(* CODESYS project FillingCappingSol_Version9.project

Project tree, tasks and I/O mapping:
  Device : CODESYS Control Win V3, 3S - Smart Software Solutions GmbH, order no. 305021, version 3.5.9.40
    application Application
      libraries: Standard, * (System)
      task MainTask (cyclic, interval t#10ms, priority 1) calls GEMMA, OutputWrite
      program F1_NormalProduction [ST]
      program D3_ProductionWithFailures [ST]
      program F2_StartingProcedure [ST]
      program F3_FinishingProcedure [ST]
      program F4_StationProducingTest [ST]
      program F5_OrderedProducingTest [ST]
      program GEMMA [ST]
      program OutputWrite [ST]
      global variables GVL
      Symbols
*)

// Device/Application/GVL
{attribute 'qualified_only'}
VAR_GLOBAL

//INPUTS
	
	//Sensors
	a0:BOOL:=FALSE;	
	a1:BOOL:=FALSE;
	b0:BOOL:=FALSE;	
	b1:BOOL:=FALSE;
	c0:BOOL:=FALSE;	
	c1:BOOL:=FALSE;
	e0:BOOL:=FALSE;	
	e1:BOOL:=FALSE;
	e2:BOOL:=FALSE;
	g0:BOOL:=FALSE;	
	g1:BOOL:=FALSE;	
	h0:BOOL:=FALSE;	
	h1:BOOL:=FALSE;	
	CP1:BOOL:=FALSE;
	CP2:BOOL:=FALSE;
	CP3:BOOL:=FALSE;	
	
	//Commands
	Mode:UINT:=0; //selector
	A:BOOL:=FALSE; //automatic
	SA:BOOL:=FALSE; //semi-automatic
	MA:BOOL:=FALSE; //manual	
	START:BOOL:=FALSE; //start PB
	PE:BOOL:=TRUE; //emergency interrupter
	STOP:BOOL:=TRUE; //stop PB	
	EM:BOOL:=FALSE; //Empty Machine
	TM:BOOL:=FALSE; //Manual Capping
	ST_:BOOL:=FALSE; //Operating Test
	CR:BOOL:=FALSE; //Capping Repaired
	OC:BOOL:=FALSE; //Operator Check
	MMC:BOOL:=FALSE; //Manual Movement Check
	
	//Semi-automatic
	Station:UINT:=0; //selector
	Station1:BOOL:=FALSE;
	Station2:BOOL:=FALSE;
	Station3:BOOL:=FALSE;
	SC:BOOL:=FALSE; //start cycle
	
	//Manual
	a_p_manual:BOOL:=FALSE; //a+
	a_m_manual:BOOL:=FALSE; //a-
	b_p_manual:BOOL:=FALSE; //b+
	b_m_manual:BOOL:=FALSE; //b-
	c_p_manual:BOOL:=FALSE; //c+
	c_m_manual:BOOL:=FALSE; //c-
	e_p_manual:BOOL:=FALSE; //e+
	g_p_manual:BOOL:=FALSE; //g+
	g_m_manual:BOOL:=FALSE; //g-
	d_p_manual:BOOL:=FALSE; //d+
	f_p_manual:BOOL:=FALSE; //f+	
	h_p_manual:BOOL:=FALSE; //h+
	h_m_manual:BOOL:=FALSE; //h-
	
	//OUTPUTS
	
	//Actuators
	a_p:BOOL:=FALSE; //a+
	a_m:BOOL:=FALSE; //a-
	b_p:BOOL:=FALSE; //b+
	b_m:BOOL:=FALSE; //b-
	c_p:BOOL:=FALSE; //c+
	c_m:BOOL:=FALSE; //c-
	e_p:BOOL:=FALSE; //e+
	g_p:BOOL:=FALSE; //g+
	g_m:BOOL:=FALSE; //g-
	d_p:BOOL:=FALSE; //d+
	f_p:BOOL:=FALSE; //f+	
	h_p:BOOL:=FALSE; //h+
	h_m:BOOL:=FALSE; //h-	
	
	//Extra
	Flag_Timer : BOOL := FALSE;
	extra2 : BOOL := FALSE;	
	Timer1 : TON;
	E_1 : BOOL := TRUE;
	E_2 : BOOL := FALSE;
	E3 : BOOL := FALSE;
	E4 : BOOL := FALSE;
	E5 : BOOL := FALSE;
	E6 : BOOL := FALSE;
	E7 : BOOL := FALSE;
	E8 : BOOL := FALSE;
	E9 : BOOL := FALSE;
	E10 : BOOL := FALSE;
	E11 : BOOL := FALSE;
	E12 : BOOL := FALSE;
	E13 : BOOL := FALSE;
	
	E20 : BOOL := TRUE;
	E21 : BOOL := FALSE;
	E22 : BOOL := FALSE;
	E23 : BOOL := FALSE;
	E24 : BOOL := FALSE;
	E25 : BOOL := FALSE;
	E26 : BOOL := FALSE;
	E27 : BOOL := FALSE;
	E28 : BOOL := FALSE;
	E29 : BOOL := FALSE;
	
	Flag_F2 : BOOL := FALSE;
	Step_Button : BOOL := FALSE;
	extra : bool := false;
END_VAR

// Device/Application/GEMMA
PROGRAM GEMMA
VAR
	State:UINT:=15;
	Flag_Entry:BOOL:=TRUE;
	RP:BOOL:=FALSE;
	
	//GEMMA states
	F1:BOOL:=FALSE;
	F2:BOOL:=FALSE;
	F3:BOOL:=FALSE;
	F4:BOOL:=FALSE;
	F5:BOOL:=FALSE;
	F6:BOOL:=FALSE;
	A1:BOOL:=FALSE;
	A2:BOOL:=FALSE;
	A3:BOOL:=FALSE;
	A4:BOOL:=FALSE;
	A5:BOOL:=FALSE;
	A6:BOOL:=FALSE;
	A7:BOOL:=FALSE;
	D1:BOOL:=FALSE;
	D2:BOOL:=FALSE;
	D3:BOOL:=FALSE;
	
	//Transitions
	T_A1_F4:BOOL:=FALSE;
	T_A1_F5:BOOL:=FALSE;
	T_A1_F2:BOOL:=FALSE;
	T_F1_D1:BOOL:=FALSE;
END_VAR

CASE State OF
	
	1:  // F1 NORMAL PRODUCTION
		IF Flag_Entry THEN
			F1:=TRUE;
			Flag_Entry:=FALSE;
		END_IF

		//Do Behavior
		F1_NormalProduction();

		T_F1_D1:=NOT GVL.PE OR F1_NormalProduction.Alarm;		
		//Exit Common Behavior
		IF T_F1_D1 OR F1_NormalProduction.T_F4 OR F1_NormalProduction.T_F5 
		OR F1_NormalProduction.T_F3 OR F1_NormalProduction.T_D3 
		OR F1_NormalProduction.T_A2 THEN
			F1:=FALSE;
			Flag_Entry:=TRUE;
		END_IF	
		//Exit Behavior
		IF T_F1_D1 THEN
			State:=7; // Transition to D1 emergency stop
			T_F1_D1:=FALSE;
		ELSIF F1_NormalProduction.T_F4 THEN
			State:=4; // Transition to F4 disordered producing test
			F1_NormalProduction.T_F4:=FALSE;
			F4_StationProducingTest.Reset:=TRUE;
 		ELSIF F1_NormalProduction.T_F5 THEN
			State:=5; // Transition to F5 ordered producing test
			F1_NormalProduction.T_F5:=FALSE;
			F5_OrderedProducingTest.Reset:=TRUE;
 		ELSIF F1_NormalProduction.T_F3 THEN
			State:=3; // Transition to F3 finishing procedure
			F1_NormalProduction.T_F3:=FALSE;
			F3_FinishingProcedure.Reset:=TRUE;
 		ELSIF F1_NormalProduction.T_D3 THEN
			State:=9; // Transition to D3 production with failure
			F1_NormalProduction.T_D3:=FALSE;
 		ELSIF F1_NormalProduction.T_A2 THEN
			State:=11; // Transition to A2 end of cycle request
			F1_NormalProduction.T_A2:=FALSE;
		END_IF
	
	2:  // F2 STARTING PROCEDURE
		
		//Entry Behavior
		IF Flag_Entry THEN
			F2:=TRUE;
			Flag_Entry:=FALSE;
		END_IF
		
		//During Behavior
		F2_StartingProcedure();
	
		//Exit Common Behavior
		IF F2_StartingProcedure.F2_DN OR NOT GVL.PE THEN
			F2:=FALSE;
			Flag_Entry:=TRUE;
		END_IF
		//Exit Behavior	
		IF NOT GVL.PE THEN
			State:=7; // Transition to D1 emergency stop
		ELSIF F2_StartingProcedure.F2_DN THEN
			State:=1; // Transition to F1 normal production
			F2_StartingProcedure.F2_DN:=FALSE;
			F1_NormalProduction.Reset:=TRUE;
		END_IF

	3:  // F3 FINISHING PROCEDURE

		//Entry Behavior
		IF Flag_Entry THEN
			F3:=TRUE;
			Flag_Entry:=FALSE;
		END_IF
		
		//Do Behavior
		F3_FinishingProcedure();

		//Exit Behavior
		IF F3_FinishingProcedure.F3_DN OR NOT GVL.PE THEN
			F3:=FALSE;
			Flag_Entry:=TRUE;
		END_IF	
		IF NOT GVL.PE THEN
			State:=7; // Transition to D1 emergency stop
		ELSIF F3_FinishingProcedure.F3_DN THEN
			State:=10; // Transition to A1 stopped at initial state
			F3_FinishingProcedure.F3_DN:=FALSE;
		END_IF
	
	4:  // F4 DISORDERED PRODUCING TEST

		//Entry Behavior
		IF Flag_Entry THEN
			F4:=TRUE;
			Flag_Entry:=FALSE;
		END_IF
		
		//Do Behavior
		F4_StationProducingTest();

		//Exit Behavior
		IF GVL.MA OR NOT GVL.PE THEN
			F4:=FALSE;
			Flag_Entry:=TRUE;
		END_IF	
		IF NOT GVL.PE THEN
			State:=7; // Transition to D1 emergency stop
		ELSIF GVL.MA THEN
			State:=15; // Transition to A6 restarting
		END_IF	

	5:  // F5 ORDERED PRODUCING TEST

		//Entry Behavior
		IF Flag_Entry THEN
			F5:=TRUE;
			Flag_Entry:=FALSE;
		END_IF
		
		//Do Behavior
		F5_OrderedProducingTest();

		//Exit Behavior
		IF F5_OrderedProducingTest.T_F1 OR F5_OrderedProducingTest.T_F4 OR NOT GVL.PE THEN
			F5:=FALSE;
			Flag_Entry:=TRUE;
		END_IF	
		IF NOT GVL.PE THEN
			State:=7; // Transition to D1 emergency stop		
		ELSIF F5_OrderedProducingTest.T_F1 THEN
			State:=1; // Transition to F1 normal production
			F5_OrderedProducingTest.T_F1:=FALSE;
			F1_NormalProduction.PreviousStateF5:=TRUE;
			F1_NormalProduction.Reset:=TRUE;
		ELSIF F5_OrderedProducingTest.T_F4 THEN
			State:=4; // Transition to F4 disordered producing test
			F5_OrderedProducingTest.T_F4:=FALSE;
			F4_StationProducingTest.Reset:=TRUE;
		END_IF
	
	6:  // F6 OPERATING TEST
	
	7:  // D1 EMERGENCY STOP

		//Entry Behavior
		IF Flag_Entry THEN
			D1:=TRUE;
			Flag_Entry:=FALSE;
		END_IF

		//Do Behavior
		RP:=GVL.h0 AND GVL.b0 AND GVL.a0 AND GVL.c0 AND NOT GVL.d_p AND NOT GVL.e_p AND NOT GVL.f_p AND GVL.g0;
		
		//Exit Behavior
		IF GVL.PE AND RP THEN
			D1:=FALSE;
			Flag_Entry:=TRUE;
			State:=14;   // Transition to A5 preparation for restarging after a failure
		END_IF	 
	
	8:  // D2 DIAGNOSIS AND TREATMENT OF FAILURES

		//Entry Behavior
		IF Flag_Entry THEN
			D2:=TRUE;
			Flag_Entry:=FALSE;
		END_IF

		//Do Behavior
		
		//Exit Behavior
		IF GVL.CR THEN
			D2:=FALSE;
			Flag_Entry:=TRUE;
			State:=14;   // Transition to A5 preparation for restarging after a failure
		END_IF	 
	
	9:  // D3 PRODUCTION WITH FAILURES

		//Entry Behavior
		IF Flag_Entry THEN
			D3:=TRUE;
			Flag_Entry:=FALSE;
		END_IF

		//Do Behavior
		D3_ProductionWithFailures();
		
		//Exit Behavior
		IF NOT GVL.TM THEN
			D3:=FALSE;
			Flag_Entry:=TRUE;
			State:=8;        // Transition to D2 diagnosis and treatment of failures
		END_IF	 
	
	10: // A1 STOPPED AT INITIAL STATE

		//Entry Behavior
		IF Flag_Entry THEN
			A1:=TRUE;
			Flag_Entry:=FALSE;
		END_IF

		//Do Behavior
		
		T_A1_F2:=GVL.START AND GVL.A;
		T_A1_F4:=GVL.START AND (GVL.MA OR GVL.ST_);
		T_A1_F5:=GVL.START AND GVL.SA;
		//Exit Behavior
		IF T_A1_F2 OR T_A1_F4 OR T_A1_F5 THEN
			A1:=FALSE;
			Flag_Entry:=TRUE;
		END_IF	 
		IF T_A1_F4 THEN 
			State:=4;     // Transition to F4 disordered producing test
			T_A1_F4:=FALSE;
			F4_StationProducingTest.Reset := TRUE;
		ELSIF T_A1_F5 THEN 
			State:=5;
			T_A1_F5:=FALSE;  // Transition to F5 ordered producing test
			F5_OrderedProducingTest.Reset:=TRUE;
		ELSIF T_A1_F2 THEN 
			State:=2;      // Transition to F2 starting procedure
			T_A1_F2:=FALSE; 
			F2_StartingProcedure.Reset:=TRUE;
		END_IF
			
	11: // A2 END OF CYCLE REQUEST

		//Entry Behavior
		IF Flag_Entry THEN
			A2:=TRUE;
			Flag_Entry:=FALSE;
		END_IF

		//Do Behavior
		RP:=GVL.h0 AND GVL.b0 AND GVL.a0 AND GVL.c0 AND NOT GVL.d_p AND NOT GVL.e_p AND NOT GVL.f_p AND GVL.g0;
		
		//Exit Behavior
		IF RP AND GVL.STOP	THEN
			A2:=FALSE;
			Flag_Entry:=TRUE;
			State:=10; // Transition to A1 stopped at initial state
			RP:=FALSE;
		END_IF	 
	
	12: // A3 STOP REQUESTED
	
	13: // A4 STOPPED AT A NOT-INITIAL STATE
	
	14: // A5 PREPARATION FOR RESTARTING AFTER A FAILURE

		//Entry Behavior
		IF Flag_Entry THEN
			A5:=TRUE;
			Flag_Entry:=FALSE;
		END_IF

		//Do Behavior
		
		//Exit Behavior
		IF GVL.OC THEN
			F1_NormalProduction.Alarm:=FALSE;
			A5:=FALSE;
			Flag_Entry:=TRUE;
			State:=15; // Transition to A6 restarting
		END_IF	 
	
	15: // A6 RESTARTING

		//Entry Behavior
		IF Flag_Entry THEN
			A6:=TRUE;
			Flag_Entry:=FALSE;
		END_IF

		//Do Behavior
		RP:=GVL.h0 AND GVL.b0 AND GVL.a0 AND GVL.c0 AND NOT GVL.d_p AND NOT GVL.e_p AND NOT GVL.f_p AND GVL.g0;
		
		//Exit Behavior
		IF RP AND GVL.MMC THEN
			A6:=FALSE;
			Flag_Entry:=TRUE;
			State:=10; // Transition to A1 stopped at initial state
			RP:=FALSE;
		END_IF	 
	
	16: // A7 STOPPING IN A NOT-INITIAL STATE

END_CASE

END_PROGRAM

// Device/Application/F1_NormalProduction
PROGRAM F1_NormalProduction
VAR
	State: INT;
	State2: INT;
	State3: INT;
	EM_MEM:BOOL:=FALSE;
	STOP_MEM:BOOL:=TRUE;
	CycleOver:BOOL:=FALSE;
END_VAR

VAR_INPUT
	Reset:BOOL:=FALSE;
	Alarm:BOOL:=FALSE;
	T_F4:BOOL:=FALSE;
	T_A2:BOOL:=FALSE;
	T_D3:BOOL:=FALSE;
	T_F5:BOOL:=FALSE;
	T_F3:BOOL:=FALSE;
	PreviousStateF5:BOOL:=FALSE;
END_VAR

IF (Reset) THEN
	Reset := FALSE;
	State:=3;
	State2:=0;
	State3:=0;
END_IF

IF PreviousStateF5 THEN
	PreviousStateF5:=FALSE;
	State:=1;
END_IF

CASE State OF
1:
	IF (GVL.b1 AND GVL.h1) THEN
		State := 2;
		CycleOver := FALSE;
	END_IF
2:
	IF (GVL.b0 AND GVL.h0) THEN
		State := 3;
	END_IF
3:
	IF (NOT GVL.CP1 OR NOT GVL.CP2 OR NOT GVL.CP3) THEN
		Alarm := TRUE;
	END_IF
	IF (NOT Alarm) THEN
		State := 4;
		State2 := 6;
		State3 := 8;
	END_IF
4:
	IF (GVL.a1) THEN
		State := 5;
	END_IF

END_CASE

CASE State2 OF
6:
	IF (GVL.c1) THEN
		State2 := 7;
	END_IF
END_CASE

CASE State3 OF
8:
	IF (GVL.g1) THEN
		State3 := 9;
	END_IF
9:
	IF (gvl.e1) THEN
		State3 := 10;
	END_IF
10:
	IF (GVL.g0) THEN
		State3 := 11;
	END_IF
11:
	IF (GVL.e2) THEN
		State3 := 12;
	END_IF
12:
		IF (GVL.a0 AND GVL.c0 AND GVL.e0) THEN
		State :=  1;
		State2 := 0;
		State3 := 0;
		CycleOver := TRUE;
	END_IF
END_CASE

//HMI Memory
IF GVL.EM OR NOT GVL.STOP THEN
	IF GVL.EM THEN
		EM_MEM:=TRUE;
	ELSIF NOT GVL.STOP THEN
		STOP_MEM:=FALSE;
	END_IF
END_IF 

//Exit Transition
IF CycleOver THEN
	IF NOT STOP_MEM THEN
		T_A2:=TRUE;
		STOP_MEM:=FALSE;
	ELSIF EM_MEM THEN
		T_F3:=TRUE;
		EM_MEM:=FALSE;	
	ELSIF GVL.MA OR GVL.ST_ THEN
		T_F4:=TRUE;
	ELSIF GVL.SA THEN
		T_F5:=TRUE;
	ELSIF GVL.TM THEN
		T_D3:=TRUE;
	END_IF
END_IF

END_PROGRAM

// Device/Application/F4_StationProducingTest
PROGRAM F4_StationProducingTest
VAR
	State: INT;
	State2: INT;
	State3: INT;
END_VAR

VAR_INPUT
		Reset: BOOL;
END_VAR

IF (Reset) THEN
	Reset := FALSE;
	State  := 1;
	State2 := 0;
	State3 := 0;
	IF NOT GVL.Station1 AND NOT GVL.Station3 THEN
		GVL.Station2:=TRUE;
	END_IF
END_IF


CASE State OF
1:
	IF (GVL.b1 AND GVL.h1) THEN
		State := 2;
	END_IF
2:
	IF (GVL.b0 AND GVL.h0) THEN
		State := 3;
	END_IF
3:
	IF (GVL.Station1 AND GVL.SC) THEN
		State := 4;
	END_IF
	IF (GVL.Station2 AND GVL.SC) THEN
		State:=0;
		State2:=6;
	END_IF
	IF (GVL.Station3 AND GVL.SC) THEN
		State:=0;
		State2:=0;
		State3:=8;
	END_IF
4:
	IF (GVL.a1) THEN
		State := 5;
	END_IF
5:
	IF (GVL.a0) THEN
		State := 13;
	END_IF
13:
		State := 3;
		State2 := 0;
		State3 := 0;
END_CASE

CASE State2 OF
6:
	IF (GVL.c1) THEN
		State2 := 7;
	END_IF
7:
	IF (GVL.c0) THEN
		State := 13;
	END_IF
END_CASE

CASE State3 OF
8:
	IF (GVL.g1) THEN
		State3 := 9;
	END_IF
9:
	IF (GVL.e1) THEN
		State3 := 10;
	END_IF
10:
	IF (GVL.g0) THEN
		State3 := 11;
	END_IF
11:
	IF (GVL.e2) THEN
		State3 := 12;
	END_IF
12:
	IF (GVL.e0) THEN
		State := 13;
	END_IF
END_CASE



IF NOT GVL.Station1 AND NOT GVL.Station3 THEN
	GVL.Station2:=TRUE;
	ELSE
		GVL.Station2 := FALSE;
END_IF

END_PROGRAM

// Device/Application/F5_OrderedProducingTest
PROGRAM F5_OrderedProducingTest
VAR
	CycleOver:BOOL:=FALSE;
	State: INT;
END_VAR
VAR_INPUT
	Reset:BOOL:=FALSE;
	T_F1:BOOL:=FALSE;
	T_F4:BOOL:=FALSE;
END_VAR

IF (Reset) THEN
	Reset := FALSE;
	State  := 1;
	CycleOver:=FALSE;
END_IF

CASE State OF 
1:	
	IF (GVL.h1 AND GVL.b1 AND GVL.Step_Button) THEN
		State := 2;
		CycleOver := FALSE;
	END_IF
2:
	IF (GVL.h0 AND GVL.b0 AND GVL.Step_Button) THEN
		State := 3;
	END_IF
3:
	IF (GVL.Step_Button AND GVL.CP1) THEN
		State := 4;
	END_IF
4:
	IF (GVL.Step_Button AND GVL.a1) THEN
		State := 5;
	END_IF
5:
	IF (GVL.Step_Button AND GVL.a0) THEN
		State := 8;
	END_IF
8:
	IF (GVL.Step_Button AND GVL.c1) THEN
		State := 9;
	END_IF
9:
	IF (GVL.Step_Button AND GVL.c0) THEN
		State := 10;
	END_IF
10:
	IF (GVL.Step_Button AND GVL.g1) THEN
		State := 11;
	END_IF
11:
	IF (GVL.Step_Button AND GVL.e1) THEN
		State := 12;
	END_IF
12:
	IF (GVL.Step_Button AND GVL.g0) THEN
		State := 13;
	END_IF
13:
	IF (GVL.Step_Button AND GVL.e2) THEN
		State := 14;
	END_IF
14:
	IF (GVL.Step_Button AND GVL.e0) THEN
		State := 1;
		CycleOver := TRUE;	
	END_IF
END_CASE

IF CycleOver THEN
	IF (GVL.A) THEN
			T_F1:=TRUE;			
	ELSIF GVL.ST_ OR GVL.MA THEN
		T_F4:=TRUE;
END_IF
END_IF

END_PROGRAM

// Device/Application/F3_FinishingProcedure
PROGRAM F3_FinishingProcedure
VAR
	State : UINT := 1;
	State2: UINT := 0;
END_VAR

VAR_INPUT
	F3_DN:BOOL:=FALSE;
	Reset:BOOL:=FALSE;
END_VAR

IF (Reset) THEN
	Reset := FALSE;
	State  := 1;
	State2 := 0;
END_IF

CASE State OF
1:
	IF (GVL.b1) THEN
		State := 2;
	END_IF	
2:
	IF (GVL.b0) THEN
		State := 3;
	END_IF
3:
	IF (NOT GVL.CP2 AND NOT GVL.CP3) THEN
		F3_DN:= TRUE;
	END_IF
	IF (GVL.CP2 AND GVL.CP3) THEN
		State := 4;
		State2 := 6;
	END_IF
	IF (NOT GVL.CP2 AND GVL.CP3) THEN
		State:= 0;
		State2 := 6;
	END_IF
4:
	IF (GVL.c1) THEN
		State := 5;
	END_IF
5:
	IF (GVL.c0 AND GVL.e0 AND State2 = 10) THEN
		State := 1;
		State2 := 0;
	END_IF
END_CASE

CASE State2 OF
6:
	IF (GVL.g1) THEN
		State2:=7;
	END_IF	
7:	
	IF (GVL.e1) THEN
		State2:=8;
	END_IF
8:
	IF (GVL.g0) THEN
		State2:=9;
	END_IF
9:
	IF (GVL.e2) THEN
		State2:=10;
	END_IF
10:
	IF (GVL.c0 AND GVL.e0 AND State=0) THEN
		State := 1;
		State2 := 0;
	END_IF
END_CASE

END_PROGRAM

// Device/Application/F2_StartingProcedure
PROGRAM F2_StartingProcedure
VAR
	State:UINT:=1;
	State2:UINT:=0;
END_VAR

VAR_INPUT
	F2_DN:BOOL:=FALSE;
	Reset:BOOL:=FALSE;
END_VAR

IF (Reset) THEN
	Reset := FALSE;
	State:=1;
	State2:=0;
END_IF

CASE State OF
1: 
	IF (GVL.h1 AND GVL.b1) THEN
		State:=2;
	END_IF;
2:
 	IF (GVL.h0 AND GVL.b0) THEN
		State:=3;
	END_IF
3:
	IF (GVL.CP1 AND GVL.CP2 AND GVL.CP3) THEN
	F2_DN := TRUE;	
	END_IF	
	IF (NOT GVL.CP1) THEN
		State := 1;
	END_IF
	IF (GVL.CP1 AND NOT GVL.CP2) THEN
		State := 4;
	END_IF
	IF(GVL.CP1 AND GVL.CP2 AND NOT GVL.CP3) THEN
		State := 6;
		State2 := 8;
	END_IF
4:
	IF(GVL.a1)THEN
		State := 5;
	END_IF
5:
	IF(GVL.a0) THEN
		State := 1;
	END_IF	
6:
	IF(GVL.a1)THEN
		State := 7;
	END_IF
7:
	IF (GVL.a0 AND GVL.c0) THEN
		State := 1;
	END_IF
END_CASE

CASE State2 OF
8:
	 IF(GVL.c1)THEN
		 State2 := 9;
	 END_IF
9:
	IF(GVL.a0 AND GVL.c0 AND State = 7)THEN
		State  := 1;
		State2 := 0;
	END_IF
END_CASE

END_PROGRAM

// Device/Application/D3_ProductionWithFailures
PROGRAM D3_ProductionWithFailures
VAR
	State:UINT:=1;
	State2:UINT:=0;
END_VAR

VAR_INPUT
	D3_DN:BOOL:=FALSE;
	Reset:BOOL:=FALSE;
END_VAR

IF (Reset) THEN
	Reset := FALSE;
	State:=1;
	State2:=0;
END_IF

CASE State OF
1:
	IF (GVL.h1 AND GVL.b1) THEN
		State := 2;
	END_IF	
2:
	IF (GVL.h0 AND GVL.b0) THEN
		State := 3;
	END_IF
3:
	IF (GVL.CP1 AND GVL.CP2) THEN
		State := 4;
		State2 := 6;
	END_IF
4:
	IF (GVL.a1) THEN
		State := 5;
	END_IF
5:
	IF (GVL.a0 AND GVL.c0 AND State2 = 7) THEN
		State := 1;
		State2 := 0;
	END_IF
END_CASE

CASE State2 OF
6:
	IF (GVL.c1) THEN
		State2 := 7;
	END_IF
END_CASE

END_PROGRAM

// Device/Application/OutputWrite
PROGRAM OutputWrite
VAR
END_VAR

GVL.a_p:=FALSE; //a+
GVL.a_m:=FALSE; //a-
GVL.b_p:=FALSE; //b+
GVL.b_m:=FALSE; //b-
GVL.c_p:=FALSE; //c+
GVL.c_m:=FALSE; //c-
GVL.e_p:=FALSE; //e+
GVL.g_p:=FALSE; //g+
GVL.g_m:=FALSE; //g-
GVL.d_p:=FALSE; //d+
GVL.h_p:=FALSE; //h+
GVL.h_m:=FALSE; //h-

//STARTING PROCEDURE ACTUATION
IF GEMMA.A6 THEN
	IF GVL.a_p_manual THEN
		GVL.a_p := TRUE;
	END_IF
	IF GVL.a_m_manual THEN
		GVL.a_m := TRUE;
	END_IF
	IF GVL.b_p_manual THEN
		GVL.b_p := TRUE;
	END_IF
	IF GVL.b_m_manual THEN
		GVL.b_m := TRUE;
	END_IF
	IF GVL.c_p_manual THEN
		GVL.c_p := TRUE;
	END_IF
	IF GVL.c_m_manual THEN
		GVL.c_m := TRUE;
	END_IF
	IF GVL.e_p_manual THEN
		GVL.e_p := TRUE;
	END_IF
	IF GVL.g_p_manual THEN
		GVL.g_p := TRUE;
	END_IF
	IF GVL.g_m_manual THEN
		GVL.g_m := TRUE;
	END_IF
	IF GVL.d_p_manual THEN
		GVL.d_p := TRUE;
	END_IF
	IF GVL.f_p_manual THEN
		GVL.f_p := TRUE;
		ELSE
			GVL.f_p := FALSE;
	END_IF
	IF GVL.h_p_manual THEN
		GVL.h_p := TRUE;
	END_IF
	IF GVL.h_m_manual THEN
		GVL.h_m := TRUE;
	END_IF	
END_IF


IF GEMMA.D3 THEN
CASE D3_ProductionWithFailures.State OF
1:
	GVL.h_p := TRUE;
	GVL.b_p := TRUE;
2:
	GVL.h_m := TRUE;
	GVL.b_m := TRUE;
4:
	GVL.a_p := TRUE;
5:
	GVL.a_m := TRUE;
END_CASE

CASE D3_ProductionWithFailures.State2 OF
6:
	GVL.c_p := TRUE;
	GVL.d_p := TRUE;
7:
	GVL.c_m := TRUE;
END_CASE
END_IF

IF GEMMA.F2 THEN
	CASE F2_StartingProcedure.State OF
		1: 
			GVL.h_p:=TRUE;
			GVL.b_p:=TRUE;
		2: 
			GVL.h_m:=TRUE;
			GVL.b_m:=TRUE;
		4: 
			GVL.a_p:=TRUE;
		5: 
			GVL.a_m:=TRUE;
		6: 
			GVL.a_p:=TRUE;
		7: 
			GVL.a_m:=TRUE;
	END_CASE
	
	CASE F2_StartingProcedure.State2 OF
		8: 
			GVL.c_p:=TRUE;
			GVL.d_p:=TRUE;
		9: 
			GVL.c_m:=TRUE;
	END_CASE	
END_IF

IF GEMMA.F1 THEN
	CASE F1_NormalProduction.State OF
		1:
			GVL.b_p := TRUE;
			GVL.h_p := TRUE;
		2:		
			GVL.b_m := TRUE;
			GVL.h_m := TRUE;
		4:
			GVL.a_p := TRUE;
		5:	
			GVL.a_m := TRUE;
	END_CASE
	
	CASE F1_NormalProduction.State2 OF
		6:
			GVL.c_p := TRUE;
			GVL.d_p := TRUE;
		7:
			GVL.c_m := TRUE;
	END_CASE
	
	CASE F1_NormalProduction.State3 OF
		8:
			GVL.g_p := TRUE;
		9:
			GVL.e_p := TRUE;
			GVL.f_p := TRUE;
		10:
			GVL.g_m := TRUE;
		11:
			GVL.e_p := TRUE;
		12:
			GVL.f_p := FALSE;
	END_CASE
END_IF

IF GEMMA.F3 THEN
	CASE F3_FinishingProcedure.State OF
		1:
			GVL.b_p := TRUE;
		2:
			GVL.b_m := TRUE;
		4:
			GVL.c_p := TRUE;
			GVL.d_p := TRUE;
		5:
			GVL.c_m := TRUE;	
	END_CASE
	
	CASE F3_FinishingProcedure.State2 OF
		6:
			GVL.g_p := TRUE;
		7:
			GVL.f_p := TRUE;
			GVL.e_p := TRUE;
		8:
			GVL.g_m := TRUE;
		9:
			GVL.e_p := TRUE;
		10:
			GVL.f_p := FALSE;
	END_CASE
END_IF

IF GEMMA.F4 THEN
	CASE F4_StationProducingTest.State OF
		1:
			GVL.b_p := TRUE;
			GVL.h_p := TRUE;
		2:
			GVL.b_m := TRUE;
			GVL.h_m := TRUE;
		4:
			GVL.a_p := TRUE;
		5:
			GVL.a_m := TRUE;	
	END_CASE	
	CASE F4_StationProducingTest.State2 OF
		6:
			GVL.c_p := TRUE;
			GVL.d_p := TRUE;
		7:
			GVL.c_m := TRUE;
	END_CASE
	CASE F4_StationProducingTest.State3 OF
		8:
			GVL.g_p := TRUE;
		9:
			GVL.e_p := TRUE;
			GVL.f_p := TRUE;
		10:
			GVL.g_m := TRUE;
		11:
			GVL.e_p := TRUE;
		12:
			GVL.f_p := FALSE;
	END_CASE
END_IF

IF GEMMA.F5 THEN
	CASE F5_OrderedProducingTest.State OF
		1: IF (GVL.Step_Button) THEN
			GVL.b_p := TRUE;
			GVL.h_p := TRUE;
			END_IF

		2:
			GVL.b_m := TRUE;
			GVL.h_m := TRUE;
		4:
			GVL.a_p := TRUE;
		5:
			GVL.a_m := TRUE;

		8:
			GVL.c_p := TRUE;
			GVL.d_p := TRUE;
		9:
			GVL.c_m := TRUE;
		10:
			GVL.g_p := TRUE;
		11:
			GVL.e_p := TRUE;
			GVL.f_p := TRUE;
		12:
			GVL.g_m := TRUE;
		13:
			GVL.e_p := TRUE;
		14:
			GVL.f_p := FALSE;
	END_CASE
END_IF

END_PROGRAM
